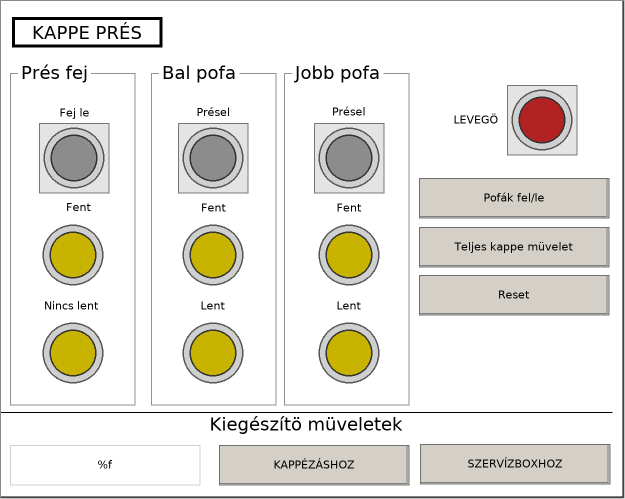
VISUALIZATION Kappe_pres  // 625x499
    Rectangle (0,0 623x497)
    GroupBox (151,65 125x340), "Bal pofa"
        Lamp1 (27,155 70x70), variable: KAPPE.bKappeBalFent, style: Lamp-Lamp1-Yellow
        Label (45,128 35x30), "Fent"
        Lamp1 (27,253 70x70), variable: KAPPE.bKappeBalLent, style: Lamp-Lamp1-Yellow
        Label (43,226 38x30), "Lent"
        PushSwitch (27,58 70x70), variable: KAPPE.bKappeBalFelLe, behaviour: TOGGLE, style: Switch-PushSwitch-Gray
        Label (37,33 51x29), "Présel"
    Button (419,178 190x40), "Pofák fel/le", input disabled if: KAPPE.bKappeBalFent<>KAPPE.bKappeJobbFent AND KAPPE.bKappeBalLent<>KAPPE.bKappeJobbLent
        OnMouseUp: execute {
            IF ((KAPPE.bKappeBalFent=TRUE) AND (KAPPE.bKappeBalLent=FALSE) AND (KAPPE.bKappeJobbFent=TRUE) AND (KAPPE.bKappeJobbLent=FALSE)) THEN
            	KAPPE.bKappeBalFelLe:=TRUE;
            	KAPPE.bKappeJobbFelLe:=TRUE;
            ELSE
            	KAPPE.bKappeBalFelLe:=FALSE;
            	KAPPE.bKappeJobbFelLe:=FALSE;
            END_IF
        }
    Button (419,227 190x40), "Teljes kappe müvelet", input disabled if: KAPPE.bKappeBalFent<>KAPPE.bKappeJobbFent AND KAPPE.bKappeBalLent<>KAPPE.bKappeJobbLent
        OnMouseUp: execute { KAPPE.s_InCommand:='START'; }
    GroupBox (284,65 125x340), "Jobb pofa"
        Lamp1 (30,155 70x70), variable: KAPPE.bKappeJobbFent, style: Lamp-Lamp1-Yellow
        Label (47,128 36x30), "Fent"
        Lamp1 (30,253 70x70), variable: KAPPE.bKappeJobbLent, style: Lamp-Lamp1-Yellow
        Label (46,226 38x30), "Lent"
        PushSwitch (30,58 70x70), variable: KAPPE.bKappeJobbFelLe, behaviour: TOGGLE, style: Switch-PushSwitch-Gray
        Label (41,32 48x30), "Présel"
    GroupBox (10,65 125x340), "Prés fej"
        Lamp1 (28,253 70x70), variable: GVL.bKappepresNincsLegalul, style: Lamp-Lamp1-Yellow
        Label (28,226 67x30), "Nincs lent"
        PushSwitch (29,58 70x70), variable: KAPPE.bKappeFelLe, behaviour: TOGGLE, style: Switch-PushSwitch-Gray
        Label (28,33 73x30), "Fej le"
        Lamp1 (28,155 70x70), variable: GVL.bKappePresFent, style: Lamp-Lamp1-Yellow
        Label (32,128 73x29), "Fent"
    RoundedRectangle (12,17 150x30)
    Label (12,18 150x30), "KAPPE PRÉS"
    Textfield (10,445 190x40), "%f", text variable: GVL.lrKappePosition
        OnMouseClick: write the text variable via VisuDialogs.Numpad, min -10000, max -1
    Button (219,445 190x40), "KAPPÉZÁSHOZ"
        OnMouseUp: execute { PISTITENGELY.lrPistiPosition:=GVL.lrKappePosition; PISTITENGELY.sPistiAxisCommand:='MOVE'; }
    Button (420,444 190x40), "SZERVÍZBOXHOZ"
        OnMouseUp: execute { PISTITENGELY.lrPistiPosition:=GVL.lrPtSzervizbox; PISTITENGELY.sPistiAxisCommand:='MOVE'; }
    Line (0,412) (612,412), "Kiegészítö müveletek"
    Group (446,85 131x70)
        PushSwitch (61,0 70x70), variable: MAIN.bLevego, behaviour: TOGGLE, style: Switch-PushSwitch-Red
        Label (0,20 55x30), "LEVEGÖ"
    Button (419,275 190x40), "Reset"
        OnMouseUp: execute { KAPPE.s_InCommand:='RESET'; }
END_VISUALIZATION

(* stored: Version 1.1.0.1, ProductVersion 3.1.4024.11
   Visu Kappe_pres: Id {5fdc2996-39f7-4f3f-8808-109eddb10bae} *)
